FUNCTION MF_Triangular : real
VAR_INPUT
	x,a,m,b:REAL;
END_VAR
VAR_OUTPUT
	error: BOOL;
END_VAR

// a < m < b
IF (a<m) AND (m<b) THEN
	IF x<=a OR x>=b THEN
		MF_Triangular:=0;
	ELSIF a<x AND x<m THEN
		MF_Triangular:=(x-a)/(m-a);
	ELSIF m<=x AND x<=b THEN
		MF_Triangular:=(b-x)/(b-m);
	END_IF
ELSE
	error:=TRUE;		
END_IF

END_FUNCTION

(* stored: Version 1.1.0.1, ProductVersion 3.1.4024.6
   POU MF_Triangular: Id {9d83b8e9-ba5c-4089-ae3d-5c67d5948293}, SpecialFunc None *)
